// TIA Portal V16 export
// export: Created 2021-11-12T13:31:39.3689808Z, ExportSetting WithDefaults, DisplayName Totally Integrated Automation Portal, DisplayVersion V16 Update 3, DisplayName TIA Portal Version Control Interface, DisplayVersion V16 Update 2, DisplayName TIA Portal Openness, DisplayVersion V16 Update 3, DisplayName SINAMICS Startdrive Advanced, DisplayVersion V16 Update 5, DisplayName SINAMICS Startdrive G130, G150, S120, S150, SINAMICS MV, S210, DisplayVersion V16 Update 5, DisplayName SINAMICS Startdrive G110M, G120, G120C, G120D, G120P, G115D, DisplayVersion V16 Update 5, DisplayName STEP 7 Professional, DisplayVersion V16 Update 3, DisplayName STEP 7 Safety, DisplayVersion V16, DisplayName WinCC UA Professional, DisplayVersion V16 Update 3
FUNCTION_BLOCK "STD_SERVO_FESTO_CMMT"   // FB43, LAD
{ S7_Optimized_Access := 'TRUE' }
VERSION : 0.1
// stored: AutoNumber true, IsIECCheckEnabled false, IsRetainMemResEnabled false, MemoryReserve 100, SetENOAutomatically false, UDAEnableTagReadback false
   VAR_INPUT
      IS_ZoneM : "UDT_Status_main";
      IS_ZoneS : "UDT_Zone_Status_specific";
      II_ModePos : Int;   // 1=Relative positioning 2=Absolute positioning 3=Not supported 4=Reference point approach 5= Set reference point 6=Traversing blocks(record mode) 7=Jog
      IB1SWLimitActive : Bool;   // 0=Software limits deactive, 1=Software limits active
      IB1GenRelDir1 : Bool;   // General release for dir 1
      IB1IntlDir1 : Bool;   // Interlock for dir 1
      IB1AutDir1 : Bool;   // Automatic command dir 1
      IB1ManDir1 : Bool;   // Manual command dir 1
      IB1GenRelDir2 : Bool;   // General release for dir 2
      IB1IntlDir2 : Bool;   // Interlock for dir 2
      IB1AutDir2 : Bool;   // Automatic command dir 2
      IB1ManDir2 : Bool;   // Manual command dir 2
      IB1AlmSupp : Bool;   // Alarms suppressed
      II_HWDSTW : HW_IO;   // Hardware identifer set point slot
      II_HWDZSW : HW_IO;   // Hardware identifer actual value slot
   END_VAR
   VAR_OUTPUT
      OS_Status : Struct
         Main : "UDT_Status_main";
         Specific : "UDT_FESTO_CMMT_Status_specific";
         Error : "UDT_Error02";
      END_STRUCT;
   END_VAR
   VAR_IN_OUT
      XS_Parameter : "UDT_FESTO_CMMT_Parameter";
      XS_Command : "UDT_FESTO_CMMT_Command";
   END_VAR
   VAR
      SS_Alarm : Struct
         CommDPRD : Bool;   // Error - Interruption of the communication to the drive: Error DPRD_DAT
         CommDPRW : Bool;   // Error - Interruption of the communication to the drive: Error DPWR_DAT
         IncorectOpMode : Bool;   // Error - Incorrect operating mode selected
         IncorParOverInputs : Bool;   // Error - Incorrect parameterization of the override inputs
         InvalidTraversBlNumber : Bool;   // Error - Invalid traversing block number
         AlarmInDrive : Bool;   // Error - Alarm message(s) in the SINAMICS drive
         SwitchOnInhibited : Bool;   // Error - Switching on inhibited of the SINAMICS drive active
         FlyingRefer : Bool;   // Error - Flying referencing could not be started
      END_STRUCT;
      SS_Warning : Struct
         PositSwitchAct : Bool;   // Warning - Positive limit switch active
         NegatSwitchAct : Bool;   // Warning - Negative limit switch active
         Warning3 : Bool;
         Warning4 : Bool;
         Warning5 : Bool;
         Warning6 : Bool;
         Warning7 : Bool;
         Warning8 : Bool;
      END_STRUCT;
      SF_SINA_POS { S7_SetPoint := 'True'} : "SINA_POS";
      SS_POS_ZSW1_Detail { S7_SetPoint := 'True'} : "UDT_FESTO_CMMT_ZSF1";
      SS_POS_ZSW2 { S7_SetPoint := 'True'} : "UDT_FESTO_CMMT_ZSW2";
      SDW_ConfigEPos : DWord;
      SB1EnableAxis : Bool;
      SB0CancelTraversing : Bool;
      SB1CollError : Bool;   // Collective error from drive
      SB1Jog1 : Bool;
      SB1Jog2 : Bool;
      SB1Positive : Bool;   // 1=Positive direction
      SB1Negative : Bool;   // 1=Negative direction
      SB1ExecuteMode : Bool;   // Comman start
      ST_AckErrPulse : TOF_TIME;   // Acknowledge error - pulse extension
   END_VAR
   VAR_TEMP
      TS_Parameter : "UDT_FESTO_CMMT_Parameter";
      TS_Command : "UDT_FESTO_CMMT_Command";
      TS_Status : Struct
         Main : "UDT_Status_main";
         Specific : "UDT_FESTO_CMMT_Status_specific";
         Error : "UDT_Error02";
      END_STRUCT;
      TB1AlmSupp : Bool;
   END_VAR
BEGIN

REGION Network 1: Clear temporary variables TS_Status
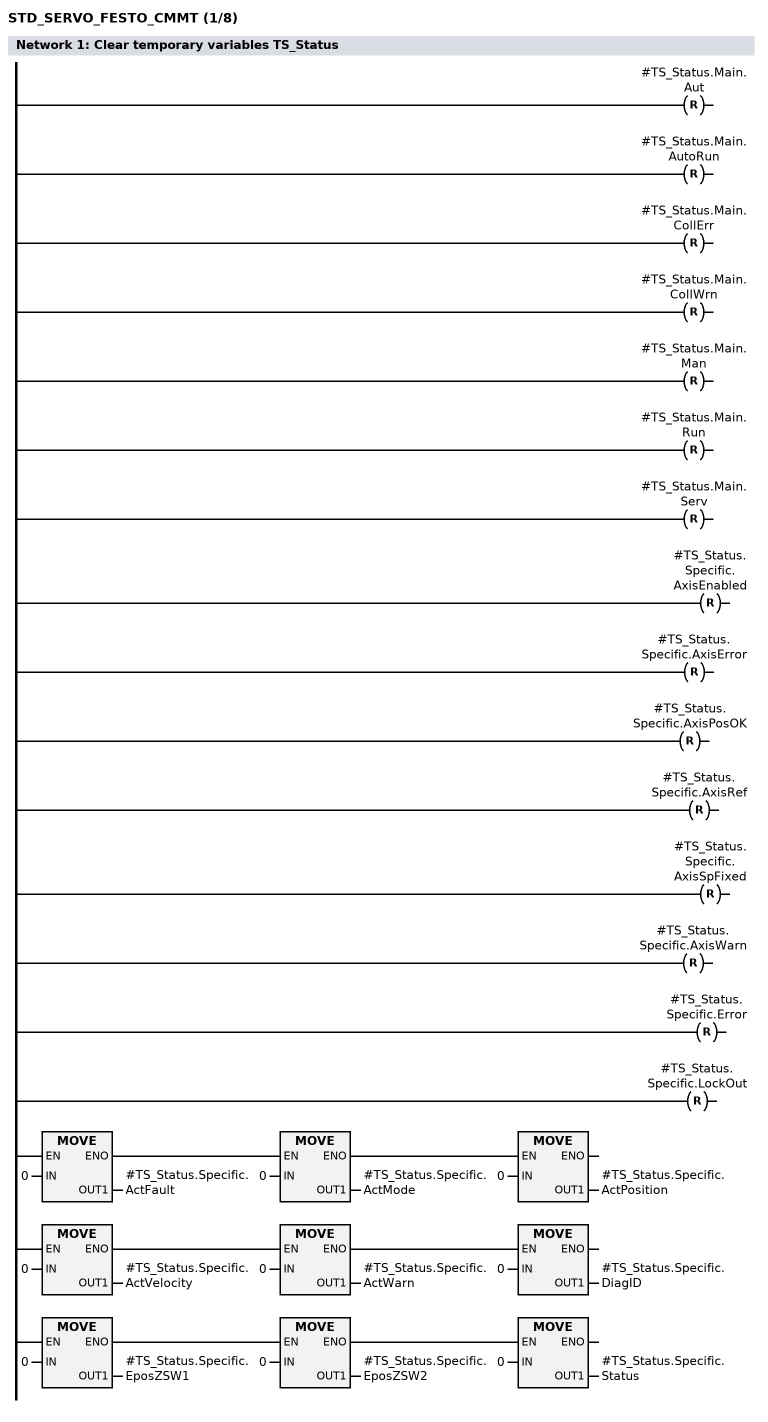
   RUNG wire#powerrail
      R_Coil( #TS_Status.Main.Aut )
   END_RUNG
   RUNG wire#powerrail
      R_Coil( #TS_Status.Main.AutoRun )
   END_RUNG
   RUNG wire#powerrail
      R_Coil( #TS_Status.Main.CollErr )
   END_RUNG
   RUNG wire#powerrail
      R_Coil( #TS_Status.Main.CollWrn )
   END_RUNG
   RUNG wire#powerrail
      R_Coil( #TS_Status.Main.Man )
   END_RUNG
   RUNG wire#powerrail
      R_Coil( #TS_Status.Main.Run )
   END_RUNG
   RUNG wire#powerrail
      R_Coil( #TS_Status.Main.Serv )
   END_RUNG
   RUNG wire#powerrail
      R_Coil( #TS_Status.Specific.AxisEnabled )
   END_RUNG
   RUNG wire#powerrail
      R_Coil( #TS_Status.Specific.AxisError )
   END_RUNG
   RUNG wire#powerrail
      R_Coil( #TS_Status.Specific.AxisPosOK )
   END_RUNG
   RUNG wire#powerrail
      R_Coil( #TS_Status.Specific.AxisRef )
   END_RUNG
   RUNG wire#powerrail
      R_Coil( #TS_Status.Specific.AxisSpFixed )
   END_RUNG
   RUNG wire#powerrail
      R_Coil( #TS_Status.Specific.AxisWarn )
   END_RUNG
   RUNG wire#powerrail
      R_Coil( #TS_Status.Specific.Error )
   END_RUNG
   RUNG wire#powerrail
      R_Coil( #TS_Status.Specific.LockOut )
   END_RUNG
   RUNG wire#powerrail
      Move(in := 0, out1 => #TS_Status.Specific.ActFault)
      Move(in := 0, out1 => #TS_Status.Specific.ActMode)
      Move(in := 0, out1 => #TS_Status.Specific.ActPosition)
   END_RUNG
   RUNG wire#powerrail
      Move(in := 0, out1 => #TS_Status.Specific.ActVelocity)
      Move(in := 0, out1 => #TS_Status.Specific.ActWarn)
      Move(in := 0, out1 => #TS_Status.Specific.DiagID)
   END_RUNG
   RUNG wire#powerrail
      Move(in := 0, out1 => #TS_Status.Specific.EposZSW1)
      Move(in := 0, out1 => #TS_Status.Specific.EposZSW2)
      Move(in := 0, out1 => #TS_Status.Specific.Status)
   END_RUNG
   // the same network as SCL:
   #TS_Status.Main.Aut := FALSE;
   #TS_Status.Main.AutoRun := FALSE;
   #TS_Status.Main.CollErr := FALSE;
   #TS_Status.Main.CollWrn := FALSE;
   #TS_Status.Main.Man := FALSE;
   #TS_Status.Main.Run := FALSE;
   #TS_Status.Main.Serv := FALSE;
   #TS_Status.Specific.AxisEnabled := FALSE;
   #TS_Status.Specific.AxisError := FALSE;
   #TS_Status.Specific.AxisPosOK := FALSE;
   #TS_Status.Specific.AxisRef := FALSE;
   #TS_Status.Specific.AxisSpFixed := FALSE;
   #TS_Status.Specific.AxisWarn := FALSE;
   #TS_Status.Specific.Error := FALSE;
   #TS_Status.Specific.LockOut := FALSE;
   #TS_Status.Specific.ActFault := 0;
   #TS_Status.Specific.ActMode := 0;
   #TS_Status.Specific.ActPosition := 0;
   #TS_Status.Specific.ActVelocity := 0;
   #TS_Status.Specific.ActWarn := 0;
   #TS_Status.Specific.DiagID := 0;
   #TS_Status.Specific.EposZSW1 := 0;
   #TS_Status.Specific.EposZSW2 := 0;
   #TS_Status.Specific.Status := 0;
END_REGION

REGION Network 2: Copy In/Out variables to temporary variables
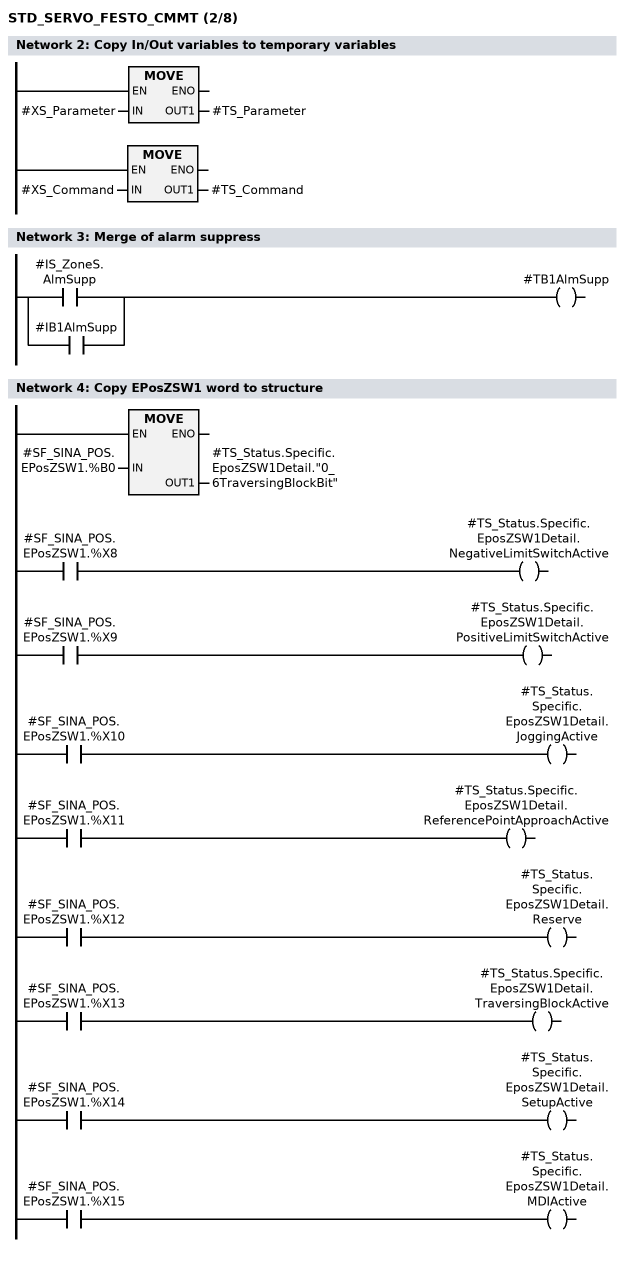
   RUNG wire#powerrail
      Move(in := #XS_Parameter, out1 => #TS_Parameter)
   END_RUNG
   RUNG wire#powerrail
      Move(in := #XS_Command, out1 => #TS_Command)
   END_RUNG
   // the same network as SCL:
   #TS_Parameter := #XS_Parameter;
   #TS_Command := #XS_Command;
END_REGION

REGION Network 3: Merge of alarm suppress
   RUNG wire#powerrail
      Contact( #IS_ZoneS.AlmSupp )
      wire#w1
      Coil( #TB1AlmSupp )
   END_RUNG
   RUNG wire#powerrail
      Contact( #IB1AlmSupp )
   END_RUNG wire#w1
   // the same network as SCL:
   #TB1AlmSupp := #IS_ZoneS.AlmSupp OR #IB1AlmSupp;
END_REGION

REGION Network 4: Copy EPosZSW1 word to structure
   RUNG wire#powerrail
      Move(in := #SF_SINA_POS.EPosZSW1.%B0, out1 => #TS_Status.Specific.EposZSW1Detail."0_6TraversingBlockBit")
   END_RUNG
   RUNG wire#powerrail
      Contact( #SF_SINA_POS.EPosZSW1.%X8 )
      Coil( #TS_Status.Specific.EposZSW1Detail.NegativeLimitSwitchActive )
   END_RUNG
   RUNG wire#powerrail
      Contact( #SF_SINA_POS.EPosZSW1.%X9 )
      Coil( #TS_Status.Specific.EposZSW1Detail.PositiveLimitSwitchActive )
   END_RUNG
   RUNG wire#powerrail
      Contact( #SF_SINA_POS.EPosZSW1.%X10 )
      Coil( #TS_Status.Specific.EposZSW1Detail.JoggingActive )
   END_RUNG
   RUNG wire#powerrail
      Contact( #SF_SINA_POS.EPosZSW1.%X11 )
      Coil( #TS_Status.Specific.EposZSW1Detail.ReferencePointApproachActive )
   END_RUNG
   RUNG wire#powerrail
      Contact( #SF_SINA_POS.EPosZSW1.%X12 )
      Coil( #TS_Status.Specific.EposZSW1Detail.Reserve )
   END_RUNG
   RUNG wire#powerrail
      Contact( #SF_SINA_POS.EPosZSW1.%X13 )
      Coil( #TS_Status.Specific.EposZSW1Detail.TraversingBlockActive )
   END_RUNG
   RUNG wire#powerrail
      Contact( #SF_SINA_POS.EPosZSW1.%X14 )
      Coil( #TS_Status.Specific.EposZSW1Detail.SetupActive )
   END_RUNG
   RUNG wire#powerrail
      Contact( #SF_SINA_POS.EPosZSW1.%X15 )
      Coil( #TS_Status.Specific.EposZSW1Detail.MDIActive )
   END_RUNG
   // the same network as SCL:
   #TS_Status.Specific.EposZSW1Detail."0_6TraversingBlockBit" := #SF_SINA_POS.EPosZSW1.%B0;
   #TS_Status.Specific.EposZSW1Detail.NegativeLimitSwitchActive := #SF_SINA_POS.EPosZSW1.%X8;
   #TS_Status.Specific.EposZSW1Detail.PositiveLimitSwitchActive := #SF_SINA_POS.EPosZSW1.%X9;
   #TS_Status.Specific.EposZSW1Detail.JoggingActive := #SF_SINA_POS.EPosZSW1.%X10;
   #TS_Status.Specific.EposZSW1Detail.ReferencePointApproachActive := #SF_SINA_POS.EPosZSW1.%X11;
   #TS_Status.Specific.EposZSW1Detail.Reserve := #SF_SINA_POS.EPosZSW1.%X12;
   #TS_Status.Specific.EposZSW1Detail.TraversingBlockActive := #SF_SINA_POS.EPosZSW1.%X13;
   #TS_Status.Specific.EposZSW1Detail.SetupActive := #SF_SINA_POS.EPosZSW1.%X14;
   #TS_Status.Specific.EposZSW1Detail.MDIActive := #SF_SINA_POS.EPosZSW1.%X15;
END_REGION

REGION Network 5: Copy EPosZSW2 word to structure
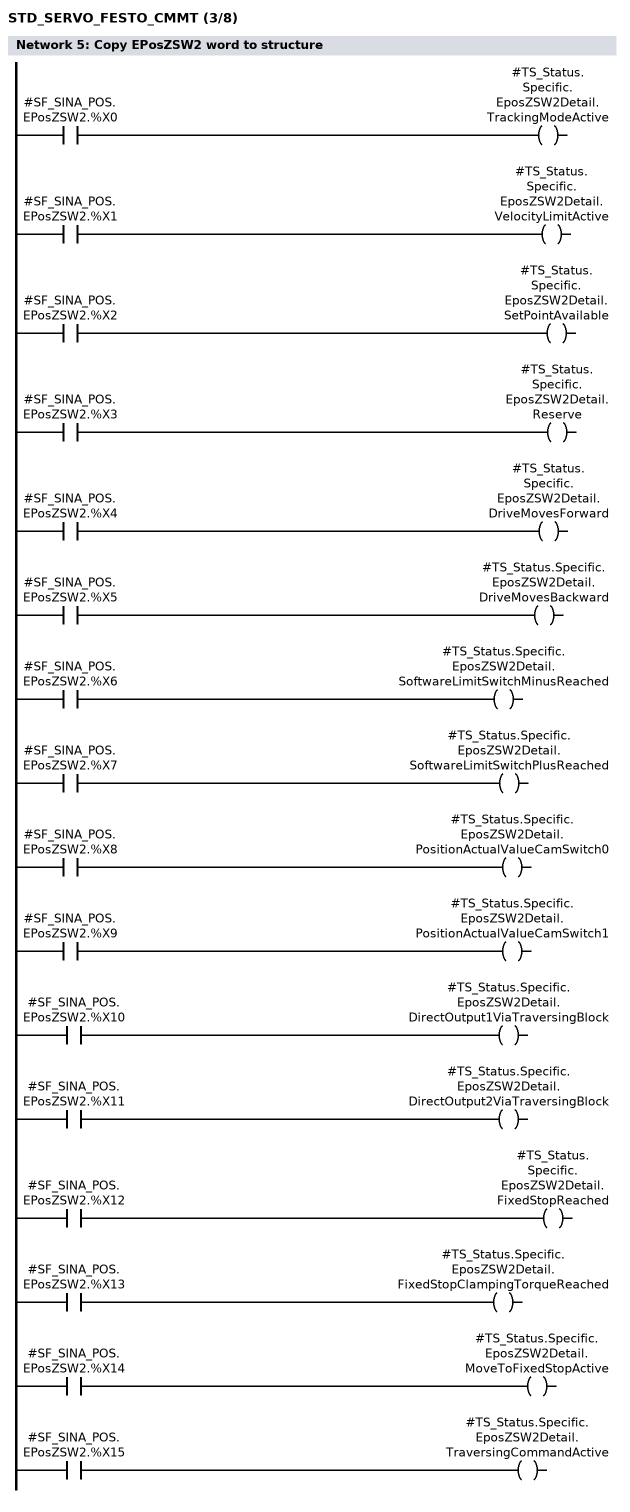
   RUNG wire#powerrail
      Contact( #SF_SINA_POS.EPosZSW2.%X0 )
      Coil( #TS_Status.Specific.EposZSW2Detail.TrackingModeActive )
   END_RUNG
   RUNG wire#powerrail
      Contact( #SF_SINA_POS.EPosZSW2.%X1 )
      Coil( #TS_Status.Specific.EposZSW2Detail.VelocityLimitActive )
   END_RUNG
   RUNG wire#powerrail
      Contact( #SF_SINA_POS.EPosZSW2.%X2 )
      Coil( #TS_Status.Specific.EposZSW2Detail.SetPointAvailable )
   END_RUNG
   RUNG wire#powerrail
      Contact( #SF_SINA_POS.EPosZSW2.%X3 )
      Coil( #TS_Status.Specific.EposZSW2Detail.Reserve )
   END_RUNG
   RUNG wire#powerrail
      Contact( #SF_SINA_POS.EPosZSW2.%X4 )
      Coil( #TS_Status.Specific.EposZSW2Detail.DriveMovesForward )
   END_RUNG
   RUNG wire#powerrail
      Contact( #SF_SINA_POS.EPosZSW2.%X5 )
      Coil( #TS_Status.Specific.EposZSW2Detail.DriveMovesBackward )
   END_RUNG
   RUNG wire#powerrail
      Contact( #SF_SINA_POS.EPosZSW2.%X6 )
      Coil( #TS_Status.Specific.EposZSW2Detail.SoftwareLimitSwitchMinusReached )
   END_RUNG
   RUNG wire#powerrail
      Contact( #SF_SINA_POS.EPosZSW2.%X7 )
      Coil( #TS_Status.Specific.EposZSW2Detail.SoftwareLimitSwitchPlusReached )
   END_RUNG
   RUNG wire#powerrail
      Contact( #SF_SINA_POS.EPosZSW2.%X8 )
      Coil( #TS_Status.Specific.EposZSW2Detail.PositionActualValueCamSwitch0 )
   END_RUNG
   RUNG wire#powerrail
      Contact( #SF_SINA_POS.EPosZSW2.%X9 )
      Coil( #TS_Status.Specific.EposZSW2Detail.PositionActualValueCamSwitch1 )
   END_RUNG
   RUNG wire#powerrail
      Contact( #SF_SINA_POS.EPosZSW2.%X10 )
      Coil( #TS_Status.Specific.EposZSW2Detail.DirectOutput1ViaTraversingBlock )
   END_RUNG
   RUNG wire#powerrail
      Contact( #SF_SINA_POS.EPosZSW2.%X11 )
      Coil( #TS_Status.Specific.EposZSW2Detail.DirectOutput2ViaTraversingBlock )
   END_RUNG
   RUNG wire#powerrail
      Contact( #SF_SINA_POS.EPosZSW2.%X12 )
      Coil( #TS_Status.Specific.EposZSW2Detail.FixedStopReached )
   END_RUNG
   RUNG wire#powerrail
      Contact( #SF_SINA_POS.EPosZSW2.%X13 )
      Coil( #TS_Status.Specific.EposZSW2Detail.FixedStopClampingTorqueReached )
   END_RUNG
   RUNG wire#powerrail
      Contact( #SF_SINA_POS.EPosZSW2.%X14 )
      Coil( #TS_Status.Specific.EposZSW2Detail.MoveToFixedStopActive )
   END_RUNG
   RUNG wire#powerrail
      Contact( #SF_SINA_POS.EPosZSW2.%X15 )
      Coil( #TS_Status.Specific.EposZSW2Detail.TraversingCommandActive )
   END_RUNG
   // the same network as SCL:
   #TS_Status.Specific.EposZSW2Detail.TrackingModeActive := #SF_SINA_POS.EPosZSW2.%X0;
   #TS_Status.Specific.EposZSW2Detail.VelocityLimitActive := #SF_SINA_POS.EPosZSW2.%X1;
   #TS_Status.Specific.EposZSW2Detail.SetPointAvailable := #SF_SINA_POS.EPosZSW2.%X2;
   #TS_Status.Specific.EposZSW2Detail.Reserve := #SF_SINA_POS.EPosZSW2.%X3;
   #TS_Status.Specific.EposZSW2Detail.DriveMovesForward := #SF_SINA_POS.EPosZSW2.%X4;
   #TS_Status.Specific.EposZSW2Detail.DriveMovesBackward := #SF_SINA_POS.EPosZSW2.%X5;
   #TS_Status.Specific.EposZSW2Detail.SoftwareLimitSwitchMinusReached := #SF_SINA_POS.EPosZSW2.%X6;
   #TS_Status.Specific.EposZSW2Detail.SoftwareLimitSwitchPlusReached := #SF_SINA_POS.EPosZSW2.%X7;
   #TS_Status.Specific.EposZSW2Detail.PositionActualValueCamSwitch0 := #SF_SINA_POS.EPosZSW2.%X8;
   #TS_Status.Specific.EposZSW2Detail.PositionActualValueCamSwitch1 := #SF_SINA_POS.EPosZSW2.%X9;
   #TS_Status.Specific.EposZSW2Detail.DirectOutput1ViaTraversingBlock := #SF_SINA_POS.EPosZSW2.%X10;
   #TS_Status.Specific.EposZSW2Detail.DirectOutput2ViaTraversingBlock := #SF_SINA_POS.EPosZSW2.%X11;
   #TS_Status.Specific.EposZSW2Detail.FixedStopReached := #SF_SINA_POS.EPosZSW2.%X12;
   #TS_Status.Specific.EposZSW2Detail.FixedStopClampingTorqueReached := #SF_SINA_POS.EPosZSW2.%X13;
   #TS_Status.Specific.EposZSW2Detail.MoveToFixedStopActive := #SF_SINA_POS.EPosZSW2.%X14;
   #TS_Status.Specific.EposZSW2Detail.TraversingCommandActive := #SF_SINA_POS.EPosZSW2.%X15;
END_REGION

REGION Network 6: Enable axis
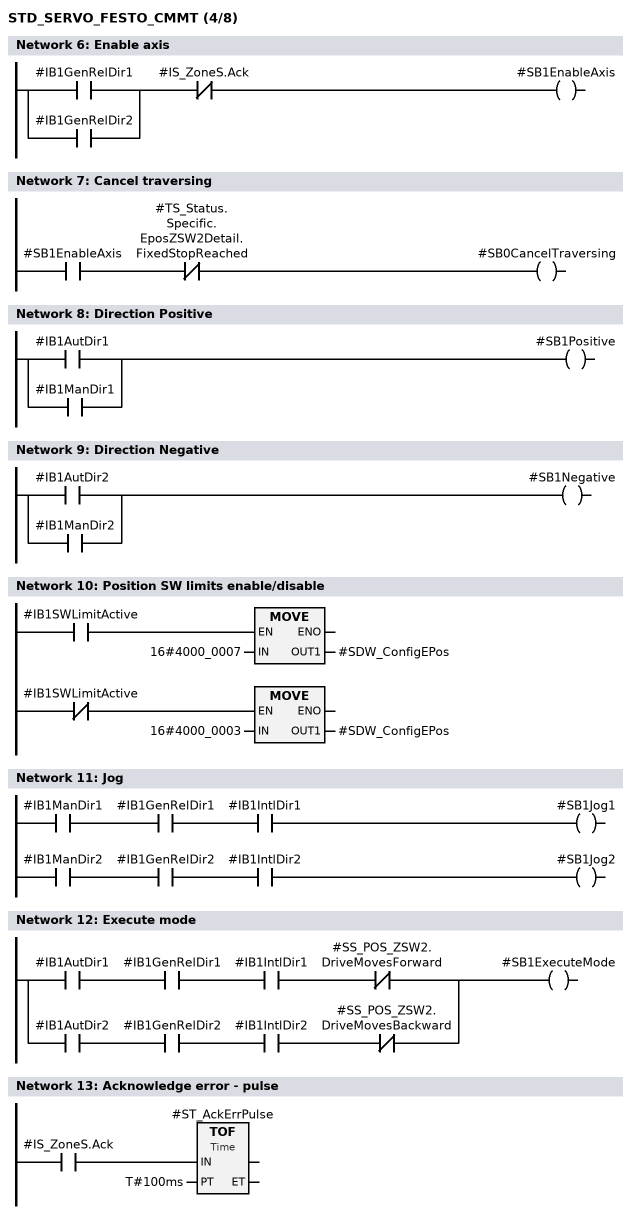
   RUNG wire#powerrail
      Contact( #IB1GenRelDir1 )
      wire#w1
      I_Contact( #IS_ZoneS.Ack )
      Coil( #SB1EnableAxis )
   END_RUNG
   RUNG wire#powerrail
      Contact( #IB1GenRelDir2 )
   END_RUNG wire#w1
   // the same network as SCL:
   #SB1EnableAxis := (#IB1GenRelDir1 OR #IB1GenRelDir2) AND NOT #IS_ZoneS.Ack;
END_REGION

REGION Network 7: Cancel traversing
   RUNG wire#powerrail
      Contact( #SB1EnableAxis )
      I_Contact( #TS_Status.Specific.EposZSW2Detail.FixedStopReached )
      Coil( #SB0CancelTraversing )
   END_RUNG
   // the same network as SCL:
   #SB0CancelTraversing := #SB1EnableAxis AND NOT #TS_Status.Specific.EposZSW2Detail.FixedStopReached;
END_REGION

REGION Network 8: Direction Positive
   RUNG wire#powerrail
      Contact( #IB1AutDir1 )
      wire#w1
      Coil( #SB1Positive )
   END_RUNG
   RUNG wire#powerrail
      Contact( #IB1ManDir1 )
   END_RUNG wire#w1
   // the same network as SCL:
   #SB1Positive := #IB1AutDir1 OR #IB1ManDir1;
END_REGION

REGION Network 9: Direction Negative
   RUNG wire#powerrail
      Contact( #IB1AutDir2 )
      wire#w1
      Coil( #SB1Negative )
   END_RUNG
   RUNG wire#powerrail
      Contact( #IB1ManDir2 )
   END_RUNG wire#w1
   // the same network as SCL:
   #SB1Negative := #IB1AutDir2 OR #IB1ManDir2;
END_REGION

REGION Network 10: Position SW limits enable/disable
   RUNG wire#powerrail
      Contact( #IB1SWLimitActive )
      Move(in := 16#4000_0007, out1 => #SDW_ConfigEPos)
   END_RUNG
   RUNG wire#powerrail
      I_Contact( #IB1SWLimitActive )
      Move(in := 16#4000_0003, out1 => #SDW_ConfigEPos)
   END_RUNG
   // the same network as SCL:
   IF #IB1SWLimitActive THEN #SDW_ConfigEPos := 16#4000_0007; END_IF;
   IF NOT #IB1SWLimitActive THEN #SDW_ConfigEPos := 16#4000_0003; END_IF;
END_REGION

REGION Network 11: Jog
   RUNG wire#powerrail
      Contact( #IB1ManDir1 )
      Contact( #IB1GenRelDir1 )
      Contact( #IB1IntlDir1 )
      Coil( #SB1Jog1 )
   END_RUNG
   RUNG wire#powerrail
      Contact( #IB1ManDir2 )
      Contact( #IB1GenRelDir2 )
      Contact( #IB1IntlDir2 )
      Coil( #SB1Jog2 )
   END_RUNG
   // the same network as SCL:
   #SB1Jog1 := #IB1ManDir1 AND #IB1GenRelDir1 AND #IB1IntlDir1;
   #SB1Jog2 := #IB1ManDir2 AND #IB1GenRelDir2 AND #IB1IntlDir2;
END_REGION

REGION Network 12: Execute mode
   RUNG wire#powerrail
      Contact( #IB1AutDir1 )
      Contact( #IB1GenRelDir1 )
      Contact( #IB1IntlDir1 )
      I_Contact( #SS_POS_ZSW2.DriveMovesForward )
      wire#w1
      Coil( #SB1ExecuteMode )
   END_RUNG
   RUNG wire#powerrail
      Contact( #IB1AutDir2 )
      Contact( #IB1GenRelDir2 )
      Contact( #IB1IntlDir2 )
      I_Contact( #SS_POS_ZSW2.DriveMovesBackward )
   END_RUNG wire#w1
   // the same network as SCL:
   #SB1ExecuteMode := (#IB1AutDir1 AND #IB1GenRelDir1 AND #IB1IntlDir1 AND NOT #SS_POS_ZSW2.DriveMovesForward) OR (#IB1AutDir2 AND #IB1GenRelDir2 AND #IB1IntlDir2 AND NOT #SS_POS_ZSW2.DriveMovesBackward);
END_REGION

REGION Network 13: Acknowledge error - pulse
   RUNG wire#powerrail
      Contact( #IS_ZoneS.Ack )
      { S7_Templates := "time_type := Time" } #ST_AckErrPulse.TOF(pt := T#100ms, et =>)
   END_RUNG
   // the same network as SCL:
   #ST_AckErrPulse(IN := #IS_ZoneS.Ack, PT := T#100ms);   // TOF
END_REGION

REGION Network 14: Control Festo
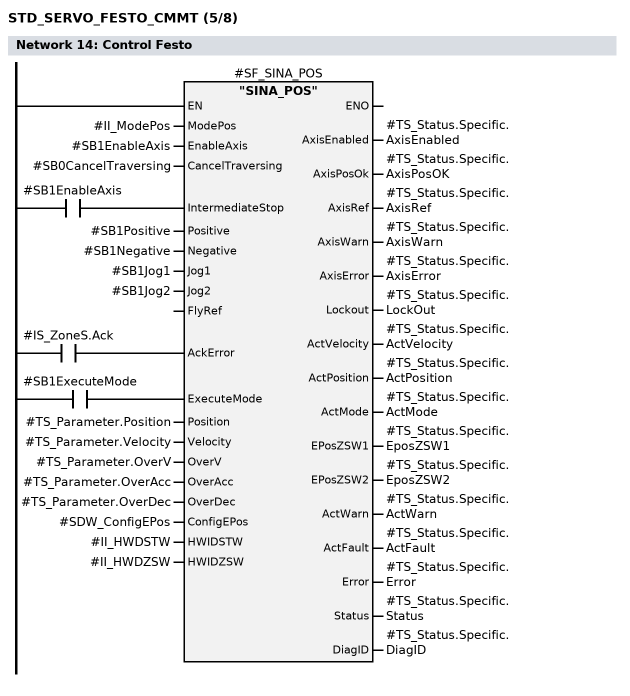
   RUNG wire#powerrail
      #SF_SINA_POS(IntermediateStop := wire#w1, AckError := wire#w2, ExecuteMode := wire#w3, ModePos := #II_ModePos, EnableAxis := #SB1EnableAxis, CancelTraversing := #SB0CancelTraversing, Positive := #SB1Positive, Negative := #SB1Negative, Jog1 := #SB1Jog1, Jog2 := #SB1Jog2, FlyRef :=, Position := #TS_Parameter.Position, Velocity := #TS_Parameter.Velocity, OverV := #TS_Parameter.OverV, OverAcc := #TS_Parameter.OverAcc, OverDec := #TS_Parameter.OverDec, ConfigEPos := #SDW_ConfigEPos, HWIDSTW := #II_HWDSTW, HWIDZSW := #II_HWDZSW, AxisEnabled => #TS_Status.Specific.AxisEnabled, AxisPosOk => #TS_Status.Specific.AxisPosOK, AxisRef => #TS_Status.Specific.AxisRef, AxisWarn => #TS_Status.Specific.AxisWarn, AxisError => #TS_Status.Specific.AxisError, Lockout => #TS_Status.Specific.LockOut, ActVelocity => #TS_Status.Specific.ActVelocity, ActPosition => #TS_Status.Specific.ActPosition, ActMode => #TS_Status.Specific.ActMode, EPosZSW1 => #TS_Status.Specific.EposZSW1, EPosZSW2 => #TS_Status.Specific.EposZSW2, ActWarn => #TS_Status.Specific.ActWarn, ActFault => #TS_Status.Specific.ActFault, Error => #TS_Status.Specific.Error, Status => #TS_Status.Specific.Status, DiagID => #TS_Status.Specific.DiagID)
   END_RUNG
   RUNG wire#powerrail
      Contact( #SB1EnableAxis )
   END_RUNG wire#w1
   RUNG wire#powerrail
      Contact( #IS_ZoneS.Ack )
   END_RUNG wire#w2
   RUNG wire#powerrail
      Contact( #SB1ExecuteMode )
   END_RUNG wire#w3
   // the same network as SCL:
   #SF_SINA_POS(ModePos := #II_ModePos,   // "SINA_POS"
                EnableAxis := #SB1EnableAxis,
                CancelTraversing := #SB0CancelTraversing,
                IntermediateStop := #SB1EnableAxis,
                Positive := #SB1Positive,
                Negative := #SB1Negative,
                Jog1 := #SB1Jog1,
                Jog2 := #SB1Jog2,
                AckError := #IS_ZoneS.Ack,
                ExecuteMode := #SB1ExecuteMode,
                Position := #TS_Parameter.Position,
                Velocity := #TS_Parameter.Velocity,
                OverV := #TS_Parameter.OverV,
                OverAcc := #TS_Parameter.OverAcc,
                OverDec := #TS_Parameter.OverDec,
                ConfigEPos := #SDW_ConfigEPos,
                HWIDSTW := #II_HWDSTW,
                HWIDZSW := #II_HWDZSW,
                AxisEnabled => #TS_Status.Specific.AxisEnabled,
                AxisPosOk => #TS_Status.Specific.AxisPosOK,
                AxisRef => #TS_Status.Specific.AxisRef,
                AxisWarn => #TS_Status.Specific.AxisWarn,
                AxisError => #TS_Status.Specific.AxisError,
                Lockout => #TS_Status.Specific.LockOut,
                ActVelocity => #TS_Status.Specific.ActVelocity,
                ActPosition => #TS_Status.Specific.ActPosition,
                ActMode => #TS_Status.Specific.ActMode,
                EPosZSW1 => #TS_Status.Specific.EposZSW1,
                EPosZSW2 => #TS_Status.Specific.EposZSW2,
                ActWarn => #TS_Status.Specific.ActWarn,
                ActFault => #TS_Status.Specific.ActFault,
                Error => #TS_Status.Specific.Error,
                Status => #TS_Status.Specific.Status,
                DiagID => #TS_Status.Specific.DiagID);
END_REGION

REGION Network 15: Errors from drive
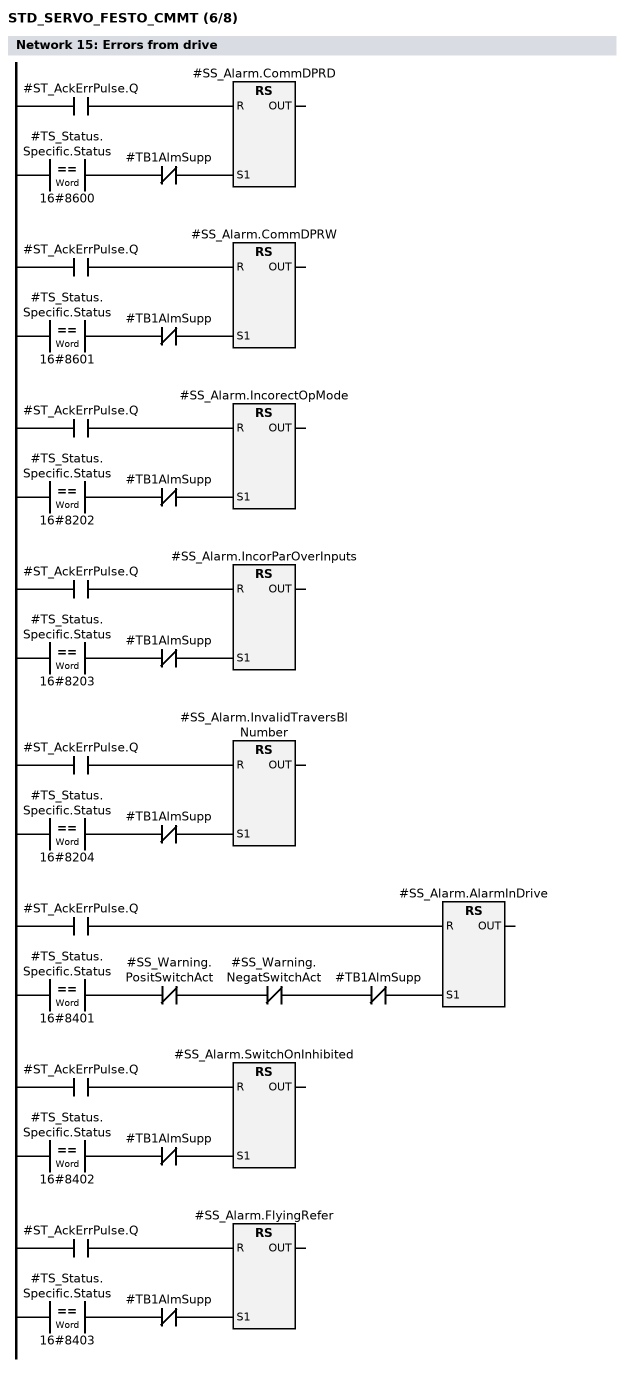
   RUNG wire#powerrail
      Contact( #ST_AckErrPulse.Q )
      S_RS(operand := #SS_Alarm.CommDPRD, s1 := wire#w1)
   END_RUNG
   RUNG wire#powerrail
      { S7_Templates := "SrcType := Word" } EQ_Contact(in1 := #TS_Status.Specific.Status, in2 := 16#8600)
      I_Contact( #TB1AlmSupp )
   END_RUNG wire#w1
   RUNG wire#powerrail
      Contact( #ST_AckErrPulse.Q )
      S_RS(operand := #SS_Alarm.CommDPRW, s1 := wire#w2)
   END_RUNG
   RUNG wire#powerrail
      { S7_Templates := "SrcType := Word" } EQ_Contact(in1 := #TS_Status.Specific.Status, in2 := 16#8601)
      I_Contact( #TB1AlmSupp )
   END_RUNG wire#w2
   RUNG wire#powerrail
      Contact( #ST_AckErrPulse.Q )
      S_RS(operand := #SS_Alarm.IncorectOpMode, s1 := wire#w3)
   END_RUNG
   RUNG wire#powerrail
      { S7_Templates := "SrcType := Word" } EQ_Contact(in1 := #TS_Status.Specific.Status, in2 := 16#8202)
      I_Contact( #TB1AlmSupp )
   END_RUNG wire#w3
   RUNG wire#powerrail
      Contact( #ST_AckErrPulse.Q )
      S_RS(operand := #SS_Alarm.IncorParOverInputs, s1 := wire#w4)
   END_RUNG
   RUNG wire#powerrail
      { S7_Templates := "SrcType := Word" } EQ_Contact(in1 := #TS_Status.Specific.Status, in2 := 16#8203)
      I_Contact( #TB1AlmSupp )
   END_RUNG wire#w4
   RUNG wire#powerrail
      Contact( #ST_AckErrPulse.Q )
      S_RS(operand := #SS_Alarm.InvalidTraversBlNumber, s1 := wire#w5)
   END_RUNG
   RUNG wire#powerrail
      { S7_Templates := "SrcType := Word" } EQ_Contact(in1 := #TS_Status.Specific.Status, in2 := 16#8204)
      I_Contact( #TB1AlmSupp )
   END_RUNG wire#w5
   RUNG wire#powerrail
      Contact( #ST_AckErrPulse.Q )
      S_RS(operand := #SS_Alarm.AlarmInDrive, s1 := wire#w6)
   END_RUNG
   RUNG wire#powerrail
      { S7_Templates := "SrcType := Word" } EQ_Contact(in1 := #TS_Status.Specific.Status, in2 := 16#8401)
      I_Contact( #SS_Warning.PositSwitchAct )
      I_Contact( #SS_Warning.NegatSwitchAct )
      I_Contact( #TB1AlmSupp )
   END_RUNG wire#w6
   RUNG wire#powerrail
      Contact( #ST_AckErrPulse.Q )
      S_RS(operand := #SS_Alarm.SwitchOnInhibited, s1 := wire#w7)
   END_RUNG
   RUNG wire#powerrail
      { S7_Templates := "SrcType := Word" } EQ_Contact(in1 := #TS_Status.Specific.Status, in2 := 16#8402)
      I_Contact( #TB1AlmSupp )
   END_RUNG wire#w7
   RUNG wire#powerrail
      Contact( #ST_AckErrPulse.Q )
      S_RS(operand := #SS_Alarm.FlyingRefer, s1 := wire#w8)
   END_RUNG
   RUNG wire#powerrail
      { S7_Templates := "SrcType := Word" } EQ_Contact(in1 := #TS_Status.Specific.Status, in2 := 16#8403)
      I_Contact( #TB1AlmSupp )
   END_RUNG wire#w8
   // the same network as SCL:
   IF #ST_AckErrPulse.Q THEN
       #SS_Alarm.CommDPRD := FALSE;   // RS flip-flop
   END_IF;
   IF (#TS_Status.Specific.Status = 16#8600) AND NOT #TB1AlmSupp THEN #SS_Alarm.CommDPRD := TRUE; END_IF;
   IF #ST_AckErrPulse.Q THEN
       #SS_Alarm.CommDPRW := FALSE;   // RS flip-flop
   END_IF;
   IF (#TS_Status.Specific.Status = 16#8601) AND NOT #TB1AlmSupp THEN #SS_Alarm.CommDPRW := TRUE; END_IF;
   IF #ST_AckErrPulse.Q THEN
       #SS_Alarm.IncorectOpMode := FALSE;   // RS flip-flop
   END_IF;
   IF (#TS_Status.Specific.Status = 16#8202) AND NOT #TB1AlmSupp THEN
       #SS_Alarm.IncorectOpMode := TRUE;
   END_IF;
   IF #ST_AckErrPulse.Q THEN
       #SS_Alarm.IncorParOverInputs := FALSE;   // RS flip-flop
   END_IF;
   IF (#TS_Status.Specific.Status = 16#8203) AND NOT #TB1AlmSupp THEN
       #SS_Alarm.IncorParOverInputs := TRUE;
   END_IF;
   IF #ST_AckErrPulse.Q THEN
       #SS_Alarm.InvalidTraversBlNumber := FALSE;   // RS flip-flop
   END_IF;
   IF (#TS_Status.Specific.Status = 16#8204) AND NOT #TB1AlmSupp THEN
       #SS_Alarm.InvalidTraversBlNumber := TRUE;
   END_IF;
   IF #ST_AckErrPulse.Q THEN
       #SS_Alarm.AlarmInDrive := FALSE;   // RS flip-flop
   END_IF;
   IF (#TS_Status.Specific.Status = 16#8401) AND NOT #SS_Warning.PositSwitchAct AND NOT #SS_Warning.NegatSwitchAct AND NOT #TB1AlmSupp THEN
       #SS_Alarm.AlarmInDrive := TRUE;
   END_IF;
   IF #ST_AckErrPulse.Q THEN
       #SS_Alarm.SwitchOnInhibited := FALSE;   // RS flip-flop
   END_IF;
   IF (#TS_Status.Specific.Status = 16#8402) AND NOT #TB1AlmSupp THEN
       #SS_Alarm.SwitchOnInhibited := TRUE;
   END_IF;
   IF #ST_AckErrPulse.Q THEN
       #SS_Alarm.FlyingRefer := FALSE;   // RS flip-flop
   END_IF;
   IF (#TS_Status.Specific.Status = 16#8403) AND NOT #TB1AlmSupp THEN #SS_Alarm.FlyingRefer := TRUE; END_IF;
END_REGION

REGION Network 16: Warning from drive
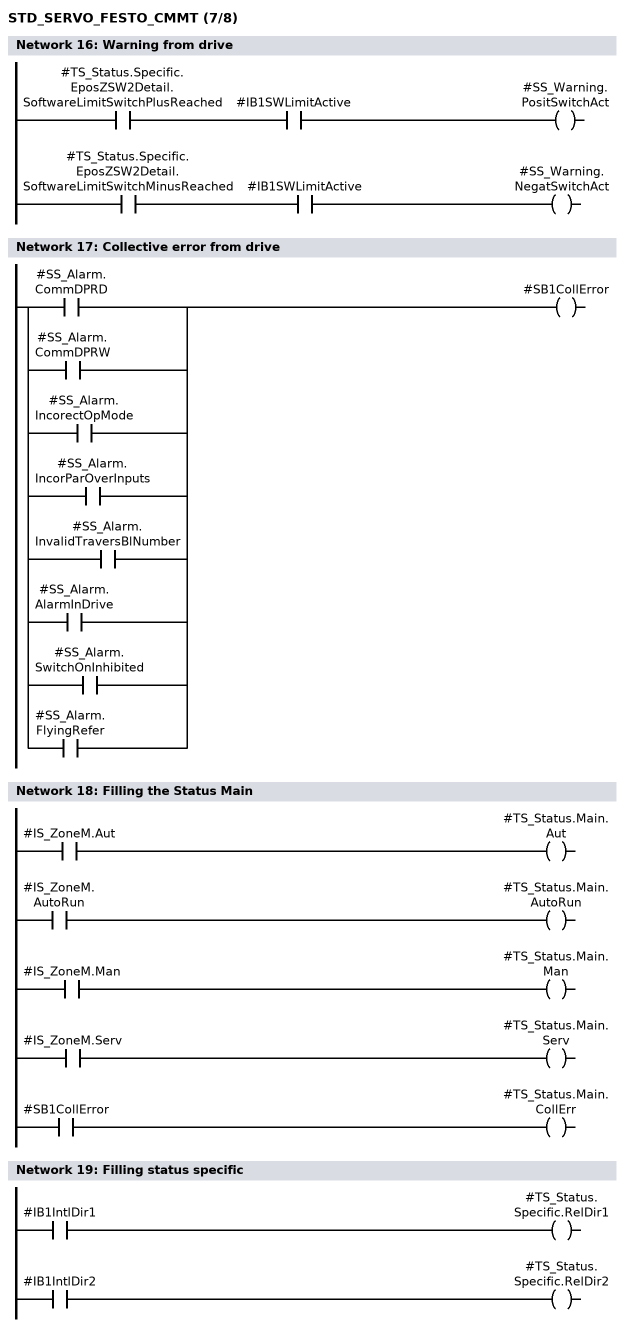
   RUNG wire#powerrail
      Contact( #TS_Status.Specific.EposZSW2Detail.SoftwareLimitSwitchPlusReached )
      Contact( #IB1SWLimitActive )
      Coil( #SS_Warning.PositSwitchAct )
   END_RUNG
   RUNG wire#powerrail
      Contact( #TS_Status.Specific.EposZSW2Detail.SoftwareLimitSwitchMinusReached )
      Contact( #IB1SWLimitActive )
      Coil( #SS_Warning.NegatSwitchAct )
   END_RUNG
   // the same network as SCL:
   #SS_Warning.PositSwitchAct := #TS_Status.Specific.EposZSW2Detail.SoftwareLimitSwitchPlusReached AND #IB1SWLimitActive;
   #SS_Warning.NegatSwitchAct := #TS_Status.Specific.EposZSW2Detail.SoftwareLimitSwitchMinusReached AND #IB1SWLimitActive;
END_REGION

REGION Network 17: Collective error from drive
   RUNG wire#powerrail
      Contact( #SS_Alarm.CommDPRD )
      wire#w1
      Coil( #SB1CollError )
   END_RUNG
   RUNG wire#powerrail
      Contact( #SS_Alarm.CommDPRW )
   END_RUNG wire#w1
   RUNG wire#powerrail
      Contact( #SS_Alarm.IncorectOpMode )
   END_RUNG wire#w1
   RUNG wire#powerrail
      Contact( #SS_Alarm.IncorParOverInputs )
   END_RUNG wire#w1
   RUNG wire#powerrail
      Contact( #SS_Alarm.InvalidTraversBlNumber )
   END_RUNG wire#w1
   RUNG wire#powerrail
      Contact( #SS_Alarm.AlarmInDrive )
   END_RUNG wire#w1
   RUNG wire#powerrail
      Contact( #SS_Alarm.SwitchOnInhibited )
   END_RUNG wire#w1
   RUNG wire#powerrail
      Contact( #SS_Alarm.FlyingRefer )
   END_RUNG wire#w1
   // the same network as SCL:
   #SB1CollError := #SS_Alarm.CommDPRD OR #SS_Alarm.CommDPRW OR #SS_Alarm.IncorectOpMode OR #SS_Alarm.IncorParOverInputs OR #SS_Alarm.InvalidTraversBlNumber OR #SS_Alarm.AlarmInDrive OR #SS_Alarm.SwitchOnInhibited OR #SS_Alarm.FlyingRefer;
END_REGION

REGION Network 18: Filling the Status Main
   RUNG wire#powerrail
      Contact( #IS_ZoneM.Aut )
      Coil( #TS_Status.Main.Aut )
   END_RUNG
   RUNG wire#powerrail
      Contact( #IS_ZoneM.AutoRun )
      Coil( #TS_Status.Main.AutoRun )
   END_RUNG
   RUNG wire#powerrail
      Contact( #IS_ZoneM.Man )
      Coil( #TS_Status.Main.Man )
   END_RUNG
   RUNG wire#powerrail
      Contact( #IS_ZoneM.Serv )
      Coil( #TS_Status.Main.Serv )
   END_RUNG
   RUNG wire#powerrail
      Contact( #SB1CollError )
      Coil( #TS_Status.Main.CollErr )
   END_RUNG
   // the same network as SCL:
   #TS_Status.Main.Aut := #IS_ZoneM.Aut;
   #TS_Status.Main.AutoRun := #IS_ZoneM.AutoRun;
   #TS_Status.Main.Man := #IS_ZoneM.Man;
   #TS_Status.Main.Serv := #IS_ZoneM.Serv;
   #TS_Status.Main.CollErr := #SB1CollError;
END_REGION

REGION Network 19: Filling status specific
   RUNG wire#powerrail
      Contact( #IB1IntlDir1 )
      Coil( #TS_Status.Specific.RelDir1 )
   END_RUNG
   RUNG wire#powerrail
      Contact( #IB1IntlDir2 )
      Coil( #TS_Status.Specific.RelDir2 )
   END_RUNG
   // the same network as SCL:
   #TS_Status.Specific.RelDir1 := #IB1IntlDir1;
   #TS_Status.Specific.RelDir2 := #IB1IntlDir2;
END_REGION

REGION Network 20: Alarms copy to structure
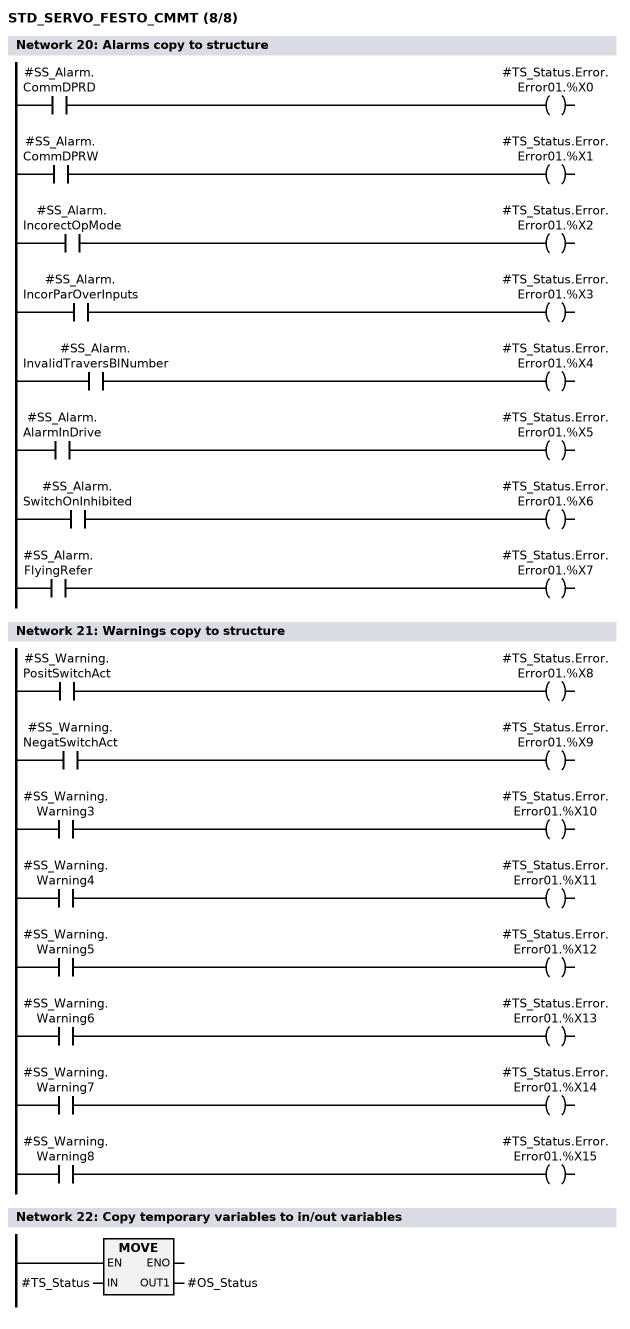
   RUNG wire#powerrail
      Contact( #SS_Alarm.CommDPRD )
      Coil( #TS_Status.Error.Error01.%X0 )
   END_RUNG
   RUNG wire#powerrail
      Contact( #SS_Alarm.CommDPRW )
      Coil( #TS_Status.Error.Error01.%X1 )
   END_RUNG
   RUNG wire#powerrail
      Contact( #SS_Alarm.IncorectOpMode )
      Coil( #TS_Status.Error.Error01.%X2 )
   END_RUNG
   RUNG wire#powerrail
      Contact( #SS_Alarm.IncorParOverInputs )
      Coil( #TS_Status.Error.Error01.%X3 )
   END_RUNG
   RUNG wire#powerrail
      Contact( #SS_Alarm.InvalidTraversBlNumber )
      Coil( #TS_Status.Error.Error01.%X4 )
   END_RUNG
   RUNG wire#powerrail
      Contact( #SS_Alarm.AlarmInDrive )
      Coil( #TS_Status.Error.Error01.%X5 )
   END_RUNG
   RUNG wire#powerrail
      Contact( #SS_Alarm.SwitchOnInhibited )
      Coil( #TS_Status.Error.Error01.%X6 )
   END_RUNG
   RUNG wire#powerrail
      Contact( #SS_Alarm.FlyingRefer )
      Coil( #TS_Status.Error.Error01.%X7 )
   END_RUNG
   // the same network as SCL:
   #TS_Status.Error.Error01.%X0 := #SS_Alarm.CommDPRD;
   #TS_Status.Error.Error01.%X1 := #SS_Alarm.CommDPRW;
   #TS_Status.Error.Error01.%X2 := #SS_Alarm.IncorectOpMode;
   #TS_Status.Error.Error01.%X3 := #SS_Alarm.IncorParOverInputs;
   #TS_Status.Error.Error01.%X4 := #SS_Alarm.InvalidTraversBlNumber;
   #TS_Status.Error.Error01.%X5 := #SS_Alarm.AlarmInDrive;
   #TS_Status.Error.Error01.%X6 := #SS_Alarm.SwitchOnInhibited;
   #TS_Status.Error.Error01.%X7 := #SS_Alarm.FlyingRefer;
END_REGION

REGION Network 21: Warnings copy to structure
   RUNG wire#powerrail
      Contact( #SS_Warning.PositSwitchAct )
      Coil( #TS_Status.Error.Error01.%X8 )
   END_RUNG
   RUNG wire#powerrail
      Contact( #SS_Warning.NegatSwitchAct )
      Coil( #TS_Status.Error.Error01.%X9 )
   END_RUNG
   RUNG wire#powerrail
      Contact( #SS_Warning.Warning3 )
      Coil( #TS_Status.Error.Error01.%X10 )
   END_RUNG
   RUNG wire#powerrail
      Contact( #SS_Warning.Warning4 )
      Coil( #TS_Status.Error.Error01.%X11 )
   END_RUNG
   RUNG wire#powerrail
      Contact( #SS_Warning.Warning5 )
      Coil( #TS_Status.Error.Error01.%X12 )
   END_RUNG
   RUNG wire#powerrail
      Contact( #SS_Warning.Warning6 )
      Coil( #TS_Status.Error.Error01.%X13 )
   END_RUNG
   RUNG wire#powerrail
      Contact( #SS_Warning.Warning7 )
      Coil( #TS_Status.Error.Error01.%X14 )
   END_RUNG
   RUNG wire#powerrail
      Contact( #SS_Warning.Warning8 )
      Coil( #TS_Status.Error.Error01.%X15 )
   END_RUNG
   // the same network as SCL:
   #TS_Status.Error.Error01.%X8 := #SS_Warning.PositSwitchAct;
   #TS_Status.Error.Error01.%X9 := #SS_Warning.NegatSwitchAct;
   #TS_Status.Error.Error01.%X10 := #SS_Warning.Warning3;
   #TS_Status.Error.Error01.%X11 := #SS_Warning.Warning4;
   #TS_Status.Error.Error01.%X12 := #SS_Warning.Warning5;
   #TS_Status.Error.Error01.%X13 := #SS_Warning.Warning6;
   #TS_Status.Error.Error01.%X14 := #SS_Warning.Warning7;
   #TS_Status.Error.Error01.%X15 := #SS_Warning.Warning8;
END_REGION

REGION Network 22: Copy temporary variables to in/out variables
   RUNG wire#powerrail
      Move(in := #TS_Status, out1 => #OS_Status)
   END_RUNG
   // the same network as SCL:
   #OS_Status := #TS_Status;
END_REGION

NETWORK
TITLE = Save RLO in BR bit. The BR bit helps to implement the EN/ENO mechanism for block calls.
      SET;
      SAVE;
      BE;
END_FUNCTION_BLOCK
